SYSTEM FLASHER_COMPLETE (* FLASHER in one device *)
  (* Standard: 61499-1 *)
  (* Version 0.1, 2009-03-05, JHC, Holobloc Inc., Deleted Application. *)
  (* Version 0.0, 2004-01-10, JHC, Rockwell Automation, Modified from FLASHERT_TESTD. *)
  DEVICE CTL_PANEL : FRAME_DEVICE(BOUNDS := [50,100,325,100], GRID := [1,1])
    RESOURCE RES1 : PANEL_RESOURCE
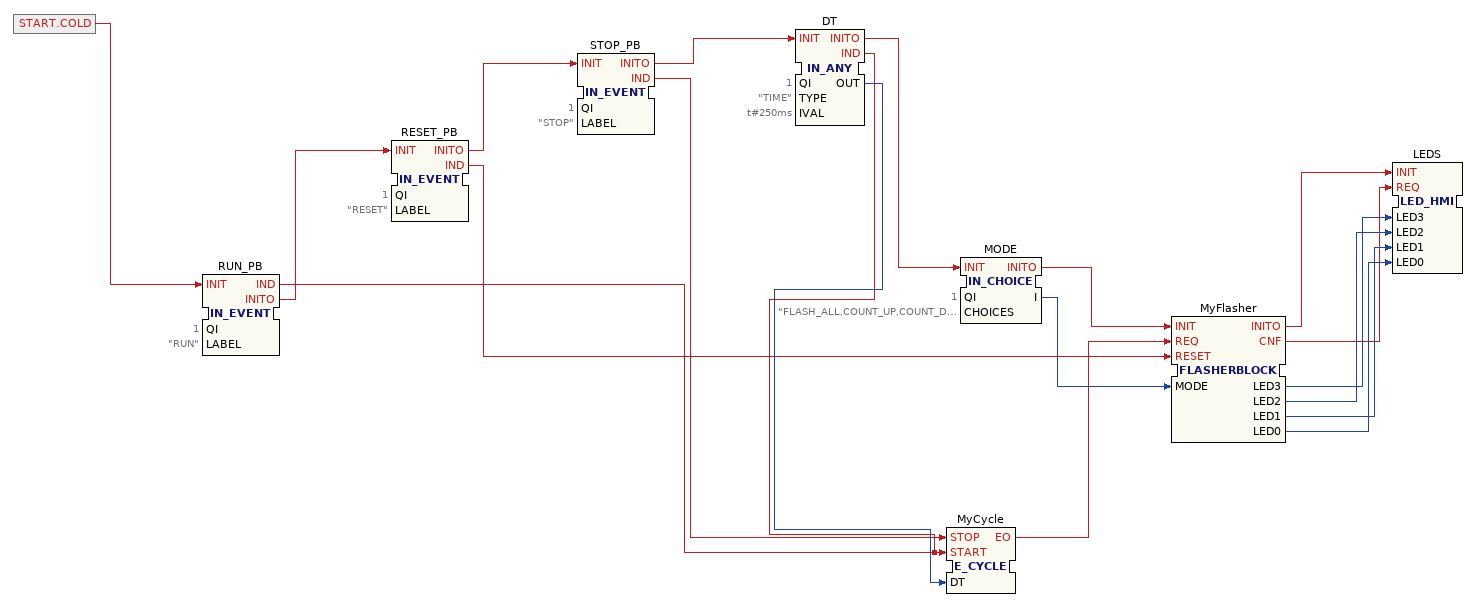
      FBS
        RUN_PB : IN_EVENT(QI := 1, LABEL := "RUN");
        STOP_PB : IN_EVENT(QI := 1, LABEL := "STOP");
        MODE : IN_CHOICE(QI := 1, CHOICES := "FLASH_ALL,COUNT_UP,COUNT_DOWN,CHASE_UP,CHASE_DOWN");
        DT : IN_ANY(QI := 1, TYPE := "TIME", IVAL := t#250ms);
        LEDS : LED_HMI;
        MyCycle : E_CYCLE;
        RESET_PB : IN_EVENT(QI := 1, LABEL := "RESET");
        MyFlasher : FLASHERBLOCK;
      END_FBS
      EVENT_CONNECTIONS
        START.COLD TO RUN_PB.INIT;
        STOP_PB.INITO TO DT.INIT;
        DT.INITO TO MODE.INIT;
        STOP_PB.IND TO MyCycle.STOP;
        DT.IND TO MyCycle.START;
        RUN_PB.IND TO MyCycle.START;
        RUN_PB.INITO TO RESET_PB.INIT;
        RESET_PB.INITO TO STOP_PB.INIT;
        MODE.INITO TO MyFlasher.INIT;
        MyFlasher.INITO TO LEDS.INIT;
        MyFlasher.CNF TO LEDS.REQ;
        MyCycle.EO TO MyFlasher.REQ;
        RESET_PB.IND TO MyFlasher.RESET;
      END_CONNECTIONS
      DATA_CONNECTIONS
        DT.OUT TO MyCycle.DT;
        MyFlasher.LED3 TO LEDS.LED3;
        MyFlasher.LED2 TO LEDS.LED2;
        MyFlasher.LED1 TO LEDS.LED1;
        MyFlasher.LED0 TO LEDS.LED0;
        MODE.I TO MyFlasher.MODE;
      END_CONNECTIONS
    END_RESOURCE
  END_DEVICE
END_SYSTEM
